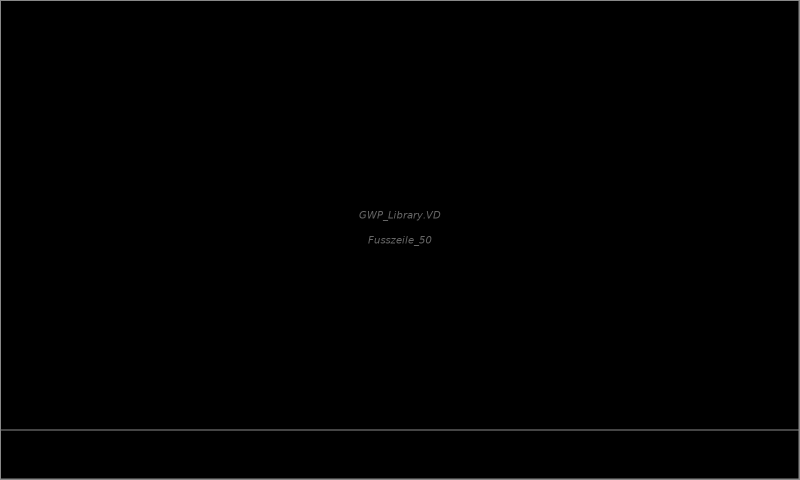
VISUALIZATION VD  // 800x480
    Frame (0,0 800x430)
        shows GWP_Library.VD(FB_VD := Main.VD_0)
    Frame (0,0 800x480)
        shows Fusszeile_50()
END_VISUALIZATION

(* stored: Version 1.1.0.1, ProductVersion 3.1.4022.6
   Visu VD: Id {5fc76324-6b3d-49bf-b27f-867d75182e23} *)
